// TIA Portal project "TSI_LI_safety" (V15.1)

(* hardware
DEVICE "S71500/ET200MP station_1"  S7-1500 station
   slot 0: "Rail_0"  Rack  6ES7 590-1***0-0AA0
   slot 1: "PLC_1"  CPU 1516F-3 PN/DP  6ES7 516-3FN00-0AB0  V1.8
      slot 3: "CPU display_1"  6ES7591-1BA00-0AA0
DEVICE "ET 200SP station_1"  ET 200SP-Station
   slot 0: "Rack_0"  Rack  6ES5 710-8MAx1
   slot 0: "120ET2"  IM 155-6 PN HF  6ES7 155-6AU00-0CN0  V4.2
   slot 1: "121DI0"  F-DI 8x24VDC HF  6ES7 136-6BA00-0CA0  V1.0
      slot 1: "121DI0"  F-DI 8x24VDC HF
   slot 2: "123DI0"  DI 8x24VDC BA  6ES7 131-6BF00-0AA0  V1.0
      slot 1: "123DI0"  DI 8x24VDC BA
   slot 3: "124DI0"  DI 8x24VDC BA  6ES7 131-6BF00-0AA0  V1.0
      slot 1: "124DI0"  DI 8x24VDC BA
   slot 4: "125AI0"  AI 2xU ST  6ES7 134-6FB00-0BA1  V1.0
      slot 1: "125AI0"  AI 2xU ST
   slot 5: "Server module_1"  Server module  6ES7 193-6PA00-0AA0  V1.1
      slot 1: "Server module_1"  Server module
   slot 127: "BA 2xRJ45"  BA 2xRJ45  6ES7 193-6AR00-0AA0  V0.0
      slot 1: "Port_1"  X1 P1 R  6ES7 193-6AR00-0AA0  V0.0
      slot 2: "Port_2"  X1 P2 R  6ES7 193-6AR00-0AA0  V0.0
DEVICE "ET 200SP station_2"  ET 200SP-Station
   slot 0: "Rack_0"  Rack  6ES5 710-8MAx1
   slot 0: "220ET2"  IM 155-6 PN HF  6ES7 155-6AU00-0CN0  V4.2
   slot 1: "202DI0"  F-DI 8x24VDC HF  6ES7 136-6BA00-0CA0  V1.0
      slot 1: "202DI0"  F-DI 8x24VDC HF
   slot 2: "204DI0"  DI 8x24VDC ST  6ES7 131-6BF00-0BA0  V1.1
      slot 1: "204DI0"  DI 8x24VDC ST
   slot 3: "205DI0"  DI 8x24VDC ST  6ES7 131-6BF00-0BA0  V1.1
      slot 1: "205DI0"  DI 8x24VDC ST
   slot 4: "206FPM2"  F-PM-E 24VDC/8A PPM ST  6ES7 136-6PA00-0BC0  V2.0
      slot 1: "206FPM2"  F-PM-E 24VDC/8A PPM ST
   slot 5: "207DO0"  DQ 8x24VDC/0.5A ST  6ES7 132-6BF00-0BA0  V1.1
      slot 1: "207DO0"  DQ 8x24VDC/0.5A ST
   slot 6: "Server module_1"  Server module  6ES7 193-6PA00-0AA0  V1.1
      slot 1: "Server module_1"  Server module
   slot 127: "BA 2xRJ45"  BA 2xRJ45  6ES7 193-6AR00-0AA0  V0.0
      slot 1: "Port_1"  X1 P1 R  6ES7 193-6AR00-0AA0  V0.0
      slot 2: "Port_2"  X1 P2 R  6ES7 193-6AR00-0AA0  V0.0
*)

// ===== PLC "PLC_1"  CPU 1516F-3 PN/DP =====
// protected blocks, not shown: "Main_Safety_RTG1", "Main_Safety_RTG1_DB"

VAR_GLOBAL   // PLC tag table "Tags 220ET2"
   "E-Stop_Stand" AT %I12.0 : Bool;   // Emergancy stop (Measuring stand)
   "SICK" AT %I12.1 : Bool;   // SICK sensor
   "Robot_ON_feedback" AT %I12.3 : Bool;   // Robot ON relay output feedback
   "E-Stop_MC" AT %I0.0 : Bool;   // Emergancy STOP (Main cabinet)
   "PM_output" AT %Q20.0 : Bool;   // Power module output control
   "Gripper_up" AT %Q4.0 : Bool;   // Rotary table gripper UP
   "Grip_Open_1" AT %I18.0 : Bool;   // Rotary table gripper 1 OPEN
   "Grip_Open_3" AT %I18.1 : Bool;   // Rotary table gripper 3 OPEN
   "Grip_Closed_1" AT %I18.2 : Bool;   // Rotary table gripper 1 CLOSED
   "Grip_Closed_3" AT %I18.3 : Bool;   // Rotary table gripper 3 CLOSED
   "Grip_Open_2" AT %I18.4 : Bool;   // Rotary table gripper 2 OPEN
   "Grip_Closed_2" AT %I18.6 : Bool;   // Rotary table gripper 2 CLOSED
   "Grip_Up_1" AT %I19.0 : Bool;   // Rotary table gripper 1 UP
   "Grip_Up_3" AT %I19.1 : Bool;   // Rotary table gripper 3 UP
   "Grip_Down_1" AT %I19.2 : Bool;   // Rotary table gripper 1 DOWN
   "Grip_Down_3" AT %I19.3 : Bool;   // Rotary table gripper 3 DOWN
   "Grip_Up_2" AT %I19.4 : Bool;   // Rotary table gripper 2 UP
   "Grip_Down_2" AT %I19.6 : Bool;   // Rotary table gripper 2 DOWN
   "Robot_ON2" AT %Q4.1 : Bool;   // Robot safety relay 2 ON
   "Gripper_down" AT %Q4.2 : Bool;   // Rotary table gripper DOWN
   "LLT_ON" AT %Q4.3 : Bool;   // Laser ON
   "Gripper_close" AT %Q4.4 : Bool;   // Rotary table gripper CLOSE
   "Robot_ON_1" AT %Q4.6 : Bool;   // Robot safety relay 1 ON
END_VAR

VAR_GLOBAL   // PLC tag table "Tags 120ET2"
   "102F3" AT %I6.0 : Bool;   // Breaker cabinet under voltage LED
   "125B0" AT %IW8 : Int;   // Temperatuere sensor
   "102F0" AT %I6.1 : Bool;   // Breaker mains
   "102F6" AT %I6.2 : Bool;   // Breaker cabinet 230VAC sockets
   "101F5" AT %I6.3 : Bool;   // Breaker Power monitoring
   "CheckAircon" AT %I6.4 : Bool;   // Aircondition check
   "104S8" AT %I6.6 : Bool;   // Main cabinet door switch
   "102F8" AT %I7.0 : Bool;   // Breaker cabinet lights
   "106F3" AT %I7.1 : Bool;   // Motor protection S120
   "104F1" AT %I7.2 : Bool;   // Breaker VDC power
   "Fuse1" AT %I7.3 : Bool;   // Fuse module check
   "104F7" AT %I7.4 : Bool;   // Breaker aircondition
   "102F2" AT %I7.6 : Bool;   // Robot protection
END_VAR

DATA_BLOCK "TSI_LI_Datablock"   // DB2
{ S7_Optimized_Access := 'TRUE' }
VERSION : 0.1
   VAR
      Safety_ACK : Bool;   // Safety ack button WinCC
      Robot_Output_Check : Bool;
      VstupET1 : Bool;
      VstupET2 : Bool;
   END_VAR
BEGIN
END_DATA_BLOCK

ORGANIZATION_BLOCK "Main"   // OB1, LAD, ProgramCycle
TITLE = "Main Program Sweep (Cycle)"
{ S7_Optimized_Access := 'TRUE' }
VERSION : 0.1
   VAR_INPUT
      Initial_Call : Bool;   // Initial call of this OB
      Remanence : Bool;   // =True, if remanent data are available
   END_VAR
   VAR_TEMP
      Out : Bool;
   END_VAR
BEGIN

REGION Network 1: Power module output control
END_REGION
END_ORGANIZATION_BLOCK